Staubli VAL3: remGetRem.pgx

program remGetRem(string& sReturn[] (dimensions=1))
begin
  // Return current remote control state
  //
  logMsg("call remGetRem")
  if bRemControlON
    sReturn="REMOTE"
  else
    sReturn="MANUAL"
  endIf
  sReturn="GETREMOTE "+sReturn
end
